{attribute 'qualified_only'}
{attribute 'strict'}
{attribute 'to_string'}
TYPE E_3102_State : //Navitrol state
	(
		INVALID		  := 0,
		START_STATE	  := 1,
		STANDBY_STATE := 2,
		AUTO_STATE	  := 3,
		FSTOP_STATE	  := 9,
		LOAD_STATE	  := 14,
		HOLD_STATE	  := 15,
		MANUAL_STATE  := 16,
		PAUSE_STATE	  := 17
	) UDINT;
END_TYPE

(* stored: Version 1.1.0.1, ProductVersion 3.1.4026.17
   DUT E_3102_State: Id {555e105a-65b6-4bde-b534-bb12db28f4a6} *)
